FUNCTION Convert_DATE_TO_DWORD : BOOL
VAR_INPUT
	in : DATE;
	out : REFERENCE TO DWORD;
END_VAR
VAR
	converted : DWORD;
END_VAR

converted := DATE_TO_DWORD(in);

IF (DWORD_TO_DATE(converted) <> in) THEN
	RETURN;
END_IF

out := converted;
Convert_DATE_TO_DWORD := TRUE;

END_FUNCTION

(* stored: Version 1.1.0.1, ProductVersion 3.1.4024.12
   POU Convert_DATE_TO_DWORD: Id {0e6a2de9-444f-4530-a59d-b98db8f3fc11}, SpecialFunc None *)
